// §3.8b probe root: one own editable value plus one child that owns three more.
// The point of the pair is the walk — the root registers no routing code at all,
// so a test that writes a child's value proves the generic path rather than a
// hand-written override (§1.1 O1).
FUNCTION_BLOCK FB_ProbeConfigUnit EXTENDS FB_UnitBase
VAR_OUTPUT
    Child : FB_ProbeConfigCM;
END_VAR
VAR_INPUT
    CycleLimit : DINT := 100;
END_VAR

Cyclic();

METHOD Setup : BOOL
VAR_INPUT
    Name : STRING(80);
END_VAR
_M_SetName(Name);
StallTime := T#0S;
Setup := M_RegisterConfigNumber(Key := 'probe.cycleLimit',
    Item := 'StationCfg/CycleLimit', LabelKey := 'project.test.cycleLimit',
    Unit := E_EngUnit.NONE, Kind := E_ConfigKind.STATION_CFG,
    Storage := E_ConfigStorage.AS_DINT, pTarget := ADR(CycleLimit),
    Minimum := 1.0, Maximum := 1000.0, RequiresReady := FALSE);
Setup := Child.Setup(Name := CONCAT(Name, '.Child')) AND Setup;
IF Setup THEN
    Setup := _M_Register(Child);
END_IF
END_METHOD

METHOD PROTECTED _M_Dispatch
_M_SetStep(StepNo := 100, StepName := 'project.test.stepA', Awaits := 0,
    AwaitingLabel := '', TimeClass := E_TimeClass.WORK, ExpectedTime := T#0S);
END_METHOD

// Test seam. The child is reachable from outside for READING, but a nested FB
// behind an output is not an assignment target, so the owner sets it — which is
// also how a real composite would configure its own child.
METHOD M_SetChildRefuse
VAR_INPUT
    Text : STRING(255);
END_VAR
Child.RefuseText := Text;
END_METHOD

END_FUNCTION_BLOCK

(* stored: Version 1.1.0.1, ProductVersion 3.1.4024.12
   POU FB_ProbeConfigUnit: Id {4e91a730-58c6-42bd-9013-8ac25de7f146}, SpecialFunc None
   Method Setup: Id {a6d05f18-7be9-4c23-90a1-fd52b8347e06}
   Method _M_Dispatch: Id {8c37b1e4-05fa-496d-a72b-3e1d0954bc87}
   Method M_SetChildRefuse: Id {5d92e0b4-1a76-4c38-9b05-27ea41f3608d} *)
